ABB RobotStudio station: Torres.rspag

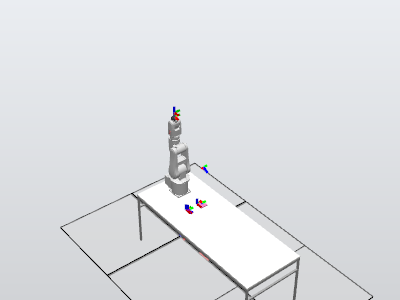
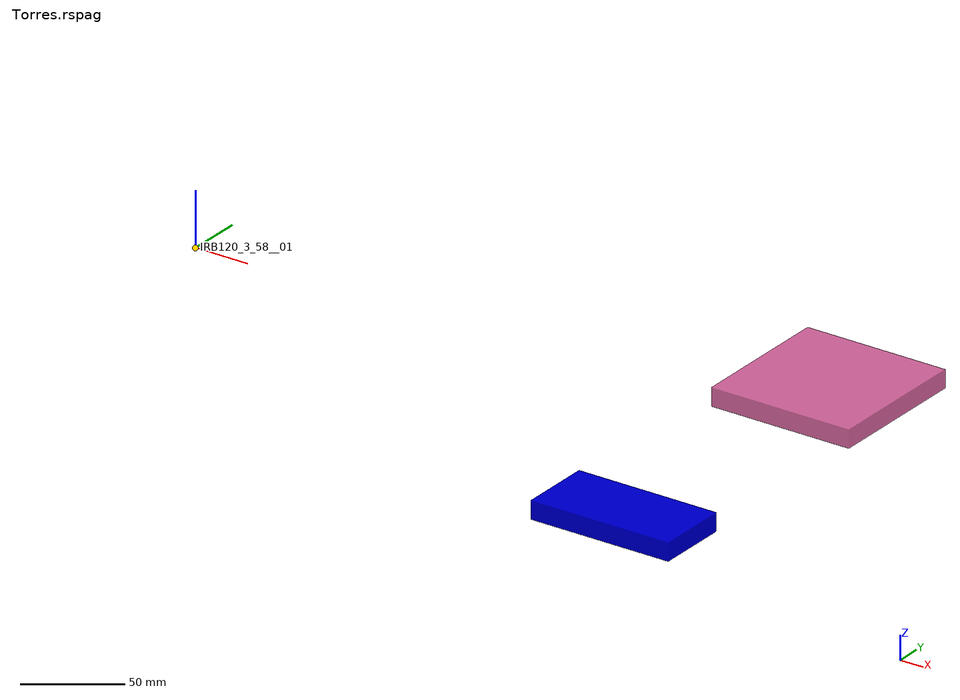
[picture v1: parts stored in the station drawn from their meshes, with robot base, taught points and paths (robot models come from the ABB library and are not in the file)]
--- station ---
Station Práctica3_inicio (saved by RobotStudio 24.3.10885.0)
Controller Controlador2, task T_ROB1: task frame (RAPID world) sits at (0, 0, 670) mm in the station
Controller Controlador2
  mechanical unit ROB_1: IRB120_3_58__01, 6 joints, base frame (0, 0, 0) mm
Layout (positions relative to the parent item):
  - TVentosa [mechanism] at (-70, 0, 1604) mm
      TCP TVentosa at (0, 0, 51.19) mm
      links: Mi_herramienta
  - LogicGate [smart component, from Components\LogicGate.rslib]
      properties: Operator=NOT; Delay=0
  - LogicGate_2 [smart component, from Components\LogicGate.rslib]
      properties: Operator=AND; Delay=0
  - IRB120_3_58__01 [mechanism, from %ABB.RobotStudio.Models.IRB120%\IRB120_3_58_G_01.rslib] at (0, 0, 670) mm; joint values [0, 0, -1.5708, 0, 0, 0] (rad or m)
  - table [part, from Libraries\e293a11e-ed86-4237-866f-a9bf8f4bd145table.rslib] at (-246.62, 300, 670) mm, rotated rx 0 ry 0 rz -90 deg
  - Base2 [part], size 80 x 80 x 10 mm
  - Base1 [part], size 80 x 40 x 10 mm
  - Detacher [smart component, from Components\Detacher.rslib]
      properties: Child=(none); KeepPosition=true
  - CollisionSensor [smart component, from Components\CollisionSensor.rslib]
      properties: Object1=TVentosa; Object2=(none); NearMiss=0.001; Part1=(none); Part2=(none); CollisionType=0
    - _sensorPart_ [part]
  - Attacher_2 [smart component, from Components\Attacher.rslib]
      properties: Parent=TVentosa; Flange=0; Child=(none); Mount=false; Offset=[0 0 0]; Orientation=[0 0 0]
  - Source_2 [smart component, from Components\Source.rslib]
      properties: Source=Pieza; Copy=(none); Parent=(none); Position=[0.34 -0.13 0.68]; Orientation=[0 0 0]; Transient=true; PhysicsBehavior=0
  - SimulationEvents_2 [smart component, from Components\SimulationEvents.rslib]
  - Pieza [part] at (340, -130, 700) mm, rotated rx 180 ry 0 rz 180 deg, size 60 x 20 x 20 mm
Attachment: TVentosa is attached to IRB120_3_58__01 / Link6
Attachment: Base2 is attached to Base1
Attachment: Base1 is attached to table
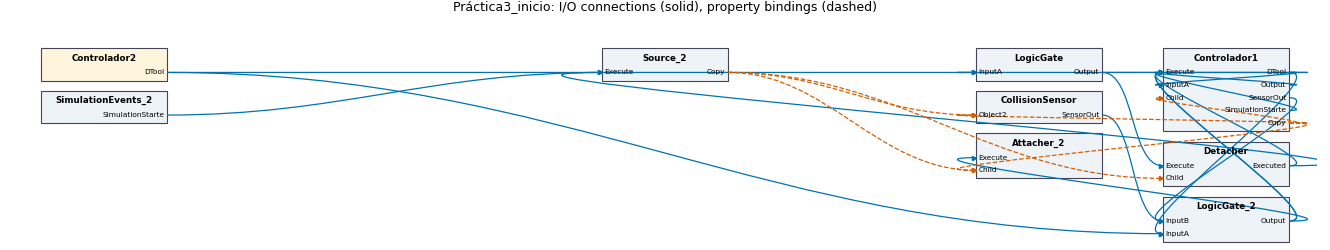
Station logic (signal -> signal, property => property):
  Controlador1.DTool -> Attacher.Execute
  Controlador1.DTool -> LogicGate_2.InputA
  LogicGate_2.Output -> Detacher.Execute
  Controlador1.DTool -> LogicGate.InputA
  LogicGate.Output -> Detacher.Execute
  CollisionSensor.SensorOut -> LogicGate_2.InputB
  Controlador1.DTool -> LogicGate_2.InputA
  LogicGate_2.Output -> Attacher.Execute
  Controlador2.DTool -> LogicGate.InputA
  LogicGate.Output -> Detacher.Execute
  Controlador2.DTool -> LogicGate_2.InputA
  LogicGate_2.Output -> Attacher.Execute
  Detacher.Executed -> Source.Execute
  SimulationEvents.SimulationStarted -> Source.Execute
  CollisionSensor.SensorOut -> LogicGate_2.InputB
  SimulationEvents_2.SimulationStarted -> Source_2.Execute
  Detacher.Executed -> Source_2.Execute
  LogicGate_2.Output -> Attacher_2.Execute
  Source.Copy => Attacher.Child
  Source.Copy => CollisionSensor.Object2
  Source.Copy => Attacher_2.Child
  Source_2.Copy => Attacher_2.Child
  Source_2.Copy => CollisionSensor.Object2
  Source_2.Copy => Detacher.Child
Targets, tools, work objects and paths stored in the station and not in the controller backup, written as RAPID:
! task T_ROB1
MODULE Module1
  PROC Path_10()
    MoveJ Target_10,v200,z100,TVentosa\WObj:=wobj0;
    MoveL Target_20,v200,fine,TVentosa\WObj:=WO_Pieza;
    MoveL Target_30,v200,z100,TVentosa\WObj:=WO_Base2;
    MoveAbsJ JHome,v1000,z100,TVentosa\WObj:=WO_Pieza;
  ENDPROC
ENDMODULE


--- Backups/Controlador2/RAPID/TASK1/PROGMOD/CalibData.mod ---
MODULE CalibData
    PERS tooldata TVentosa:=[TRUE,[[0,0,51.19],[1,0,0,0]],[0.1,[0,0,1],[1,0,0,0],0,0,0]];
    TASK PERS wobjdata WO_Pieza:=[FALSE,TRUE,"",[[300,-150,10],[1,0,0,0]],[[20,10,0],[1,0,0,0]]];
    TASK PERS wobjdata WO_Base2:=[FALSE,TRUE,"",[[300,-150,10],[1,0,0,0]],[[0,150,0],[1,0,0,0]]];
ENDMODULE

--- Backups/Controlador2/RAPID/TASK1/PROGMOD/Module1.mod ---
MODULE Module1
    CONST robtarget Target_10:=[[408.685,0,568.405],[0.5,0,0.866025404,0],[0,0,0,0],[9E+09,9E+09,9E+09,9E+09,9E+09,9E+09]];
    CONST robtarget Target_20:=[[19.999989664,10.000006428,19.999948885],[-0.000000013,0,1,0.000000005],[-1,0,-1,0],[9E+09,9E+09,9E+09,9E+09,9E+09,9E+09]];
    CONST robtarget Target_30:=[[40,40,20],[0,0,1,0],[0,0,0,0],[9E+09,9E+09,9E+09,9E+09,9E+09,9E+09]];
    CONST jointtarget JHome:=[[0,0,-90,0,0,0],[9E+09,9E+09,9E+09,9E+09,9E+09,9E+09]];

    ! Variables globales
    VAR num h;
    VAR num nueva_consigna;
    VAR num num_pieza;
    VAR num target_piezas;

    ! Procedimiento principal
    PROC main()

        ! 1. Inicializar variables y mover al robot a la posición de reposo inicial
        Initialize;
        MoveAbsJ JHome,v400,z200,TVentosa\WObj:=WO_Pieza;





            ! 2. Solicitar por consola el número de plantas
            TPReadNum nueva_consigna, "Indica la altura de la torre";
            TPErase;
            target_piezas := nueva_consigna * 4; ! Cada planta tiene 4 piezas

            ! 3. Bucle de construcción: se ejecuta hasta completar la torre o pulsar DFin
            WHILE num_pieza < target_piezas AND DFin = 0 DO

                IF DPieza = 1 THEN ! Solo avanza si hay una pieza lista en el alimentador
                    Pick Target_20, WO_Pieza;
                    Place calcula_posicion(num_pieza), WO_Base2;
                    num_pieza := num_pieza + 1;
                ENDIF



        ENDWHILE

        ! 4. Al concluir la aplicación, el manipulador vuelve a reposo
        MoveAbsJ JHome,v400,z200,TVentosa\WObj:=WO_Pieza;

    ENDPROC

    ! Rutina de inicialización
    PROC Initialize()
        h := 0;
        num_pieza := 0;
        nueva_consigna := 0;
        target_piezas := 0;
    ENDPROC

    ! Función de cálculo de la posición
    FUNC robtarget calcula_posicion(num num_pieza)
        VAR robtarget punto;
        VAR num planta;
        VAR num pos_en_planta;
        planta := num_pieza DIV 4;
        pos_en_planta := num_pieza MOD 4;
        h := planta * 40;

        TEST pos_en_planta
        CASE 0:
            punto := Offs(Target_30, 0, 20, h);
            punto.rot := Target_30.rot;
        CASE 1:
            punto := Offs(Target_30, 0, -20, h);
            punto.rot := Target_30.rot;
        CASE 2:
            punto := Offs(Target_30, 20, 0, h + 20);
            punto.rot := OrientZYX(90, 0, 180);
        CASE 3:
            punto := Offs(Target_30, -20, 0, h + 20);
            punto.rot := OrientZYX(90, 0, 180);
        ENDTEST

        RETURN punto;
    ENDFUNC

    ! Rutina para recoger la pieza
    PROC Pick(robtarget posicion, PERS wobjdata WO)
        MoveJ Offs(posicion,0,0,50),v400,z100,TVentosa\WObj:=WO;
        MoveL posicion,v300,fine,TVentosa\WObj:=WO;
        SetDO DTool,1;
        WaitTime 0.5;
        MoveL Offs(posicion,0,0,50),v300,z100,TVentosa\WObj:=WO;
    ENDPROC


    ! Rutina para dejar la pieza
    PROC Place(robtarget posicion, PERS wobjdata WO)
        MoveJ Offs(posicion,0,0,50),v400,fine,TVentosa\WObj:=WO;
        MoveL posicion,v300,fine,TVentosa\WObj:=WO;
        SetDO DTool,0;
        WaitTime 0.5;
        MoveL Offs(posicion,0,0,50),v300,fine,TVentosa\WObj:=WO;
    ENDPROC

ENDMODULE

--- Backups/Controlador2/SYSPAR/EIO.cfg ---
EIO:CFG_1.0:6:1::
#
EIO_SIGNAL:

      -Name "DFin" -SignalType "DI"

      -Name "DTool" -SignalType "DO"

      -Name "DPieza" -SignalType "DI"
